FUNCTION_BLOCK Mc2AxisPTP_HMI EXTENDS HmiFunction
VAR
	Axis : I_Mc2Axis_PTP;
	{ attribute 'TcHmiSymbol.AddSymbol' }
	{ attribute 'TcHmiSymbol.AddSymbol.UserGroups' := '__SystemAdministrators,Admin' }
	AxisPTP_HMI : ST_AxisPTP_HMI;
END_VAR

PROPERTY ControlObject : I_Base
SET
__QueryInterface(ControlObject,Axis);
END_SET
END_PROPERTY

METHOD CyclicLogic
VAR_INST
	EnableRT	   : R_TRIG;
	DisableRT	   : R_TRIG;
	StopRT		   : R_TRIG;
	HomeRT		   : R_TRIG;
	ResetRT		   : R_TRIG;
	MoveAbsoluteRT : R_TRIG;
	MoveModuloRT   : R_TRIG;
	MoveRelativeRT : R_TRIG;
	MoveVelocityRT : R_TRIG;
END_VAR
IF Axis = 0 THEN
	RETURN;
END_IF

AxisPTP_HMI.HmiEnabled				  := Enabled;
AxisPTP_HMI.ActualAcceleration		  := Axis.ActualAcceleration;
AxisPTP_HMI.ActualPosition			  := Axis.ActualPosition;
AxisPTP_HMI.ActualPositionModulo	  := Axis.ActualPositionModulo;
AxisPTP_HMI.ActualTorque			  := Axis.ActualTorque;
AxisPTP_HMI.ActualVelocity			  := Axis.ActualVelocity;
AxisPTP_HMI.Busy					  := Axis.Busy;
AxisPTP_HMI.Error					  := Axis.Error;
AxisPTP_HMI.ErrorId					  := Axis.ErrorId;
AxisPTP_HMI.Name					  := Axis.Name;
AxisPTP_HMI.Status.Coupled			  := Axis.Axis.Status.Coupled;
AxisPTP_HMI.Status.Disabled			  := Axis.Axis.Status.Disabled;
AxisPTP_HMI.Status.SynchronizedMotion := Axis.Axis.Status.SynchronizedMotion;

// HMI Commands
StopRT(CLK := AxisPTP_HMI.Stop.Active);
IF StopRT.Q THEN
	IF AxisPTP_HMI.Stop.Permissive.OK THEN
		Axis.Stop();
	END_IF
END_IF

ResetRT(CLK := AxisPTP_HMI.Reset.Active);
IF ResetRT.Q THEN
	IF AxisPTP_HMI.Reset.Permissive.OK THEN
		Axis.Reset();
	END_IF
END_IF

IF Enabled THEN
	EnableRT(CLK := AxisPTP_HMI.Enable.Active);
	IF EnableRT.Q THEN
		IF AxisPTP_HMI.Enable.Permissive.OK THEN
			Axis.Enable();
		END_IF
	END_IF

	DisableRT(CLK := AxisPTP_HMI.Disable.Active);
	IF DisableRT.Q THEN
		IF AxisPTP_HMI.Disable.Permissive.OK THEN
			Axis.Disable();
		END_IF
	END_IF

	IF AxisPTP_HMI.JogBackwardSlow.Active THEN
		IF AxisPTP_HMI.JogBackwardSlow.Permissive.OK THEN
			Axis.JogMode := E_JogMode.MC_JOGMODE_STANDARD_SLOW;
			Axis.Jog(JogForward := FALSE, JogBackwards := TRUE);
		END_IF
	ELSIF AxisPTP_HMI.JogForwardSlow.Active THEN
		Axis.JogMode := E_JogMode.MC_JOGMODE_STANDARD_SLOW;
		Axis.Jog(JogForward := TRUE, JogBackwards := FALSE);
	ELSIF AxisPTP_HMI.JogBackwardFast.Active THEN
		Axis.JogMode := E_JogMode.MC_JOGMODE_STANDARD_FAST;
		Axis.Jog(JogForward := FALSE, JogBackwards := TRUE);
	ELSIF AxisPTP_HMI.JogForwardFast.Active THEN
		Axis.JogMode := E_JogMode.MC_JOGMODE_STANDARD_FAST;
		Axis.Jog(JogForward := TRUE, JogBackwards := FALSE);
	ELSE
		Axis.JogMode := E_JogMode.MC_JOGMODE_STANDARD_SLOW;
		Axis.Jog(JogForward := FALSE, JogBackwards := FALSE);
	END_IF

	HomeRT(CLK := AxisPTP_HMI.Home.Active);
	IF HomeRT.Q THEN
		IF AxisPTP_HMI.Home.Permissive.OK THEN
			Axis.Home();
		END_IF
	END_IF

	MoveAbsoluteRT(CLK := AxisPTP_HMI.MoveAbsolute.Active);
	IF MoveAbsoluteRT.Q THEN
		IF AxisPTP_HMI.MoveAbsolute.Permissive.OK THEN
			Axis.MoveAbsolute(AxisPTP_HMI.TargetPosition);
		END_IF
	END_IF

	MoveModuloRT(CLK := AxisPTP_HMI.MoveModulo.Active);
	IF MoveModuloRT.Q THEN
		IF AxisPTP_HMI.MoveModulo.Permissive.OK THEN
			Axis.MoveModulo(AxisPTP_HMI.TargetPosition);
		END_IF
	END_IF

	MoveRelativeRT(CLK := AxisPTP_HMI.MoveRelative.Active);
	IF MoveRelativeRT.Q THEN
		IF AxisPTP_HMI.MoveRelative.Permissive.OK THEN
			Axis.MoveRelative(AxisPTP_HMI.TargetDistance);
		END_IF
	END_IF

	MoveVelocityRT(CLK := AxisPTP_HMI.MoveVelocity.Active);
	IF MoveVelocityRT.Q THEN
		IF AxisPTP_HMI.MoveVelocity.Permissive.OK THEN
			Axis.MoveVelocity(AxisPTP_HMI.TargetVelocity);
		END_IF
	END_IF
END_IF
END_METHOD

PROPERTY DisablePermissive : I_Permissive
GET
DisablePermissive := AxisPTP_HMI.Disable.Permissive;
END_GET
END_PROPERTY

PROPERTY EnablePermissive : I_Permissive
GET
EnablePermissive := AxisPTP_HMI.Enable.Permissive;
END_GET
END_PROPERTY

(*FB_Init is always available implicitly and it is used primarily for initialization.
The return value is not evaluated. For a specific influence, you can also declare the
methods explicitly and provide additional code there with the standard initialization
code. You can evaluate the return value.*)
METHOD FB_Init : BOOL
VAR_INPUT
	(* TRUE: the retain variables are initialized (reset warm / reset cold)*)
	bInitRetains : BOOL;

	(* TRUE: the instance will be copied to the copy code afterward (online change)   *)
	bInCopyCode : BOOL;
	Name		: T_MaxString;
	Axis		: I_Mc2Axis_PTP;
	Unit		: STRING;
END_VAR
THIS^.Axis		 := Axis;
ControlType		 := 'AxisPTP';
LinkObject		 := 'AxisPTP_HMI';
AxisPTP_HMI.Unit := Unit;
END_METHOD

PROPERTY HomePermissive : I_Permissive
GET
HomePermissive := AxisPTP_HMI.Home.Permissive;
END_GET
END_PROPERTY

PROPERTY JogBackwardFastPermissive : I_Permissive
GET
JogBackwardFastPermissive := AxisPTP_HMI.JogBackwardFast.Permissive;
END_GET
END_PROPERTY

PROPERTY JogBackwardSlowPermissive : I_Permissive
GET
JogBackwardSlowPermissive := AxisPTP_HMI.JogBackwardSlow.Permissive;
END_GET
END_PROPERTY

PROPERTY JogForwardFastPermissive : I_Permissive
GET
JogForwardFastPermissive := AxisPTP_HMI.JogForwardFast.Permissive;
END_GET
END_PROPERTY

PROPERTY JogForwardSlowPermissive : I_Permissive
GET
JogForwardSlowPermissive := AxisPTP_HMI.JogForwardSlow.Permissive;
END_GET
END_PROPERTY

PROPERTY MoveAbsolutePermissive : I_Permissive
GET
MoveAbsolutePermissive := AxisPTP_HMI.MoveAbsolute.Permissive;
END_GET
END_PROPERTY

PROPERTY MoveModuloPermissive : I_Permissive
GET
MoveModuloPermissive := AxisPTP_HMI.MoveModulo.Permissive;
END_GET
END_PROPERTY

PROPERTY MoveRelativePermissive : I_Permissive
GET
MoveRelativePermissive := AxisPTP_HMI.MoveRelative.Permissive;
END_GET
END_PROPERTY

PROPERTY MoveVelocityPermissive : I_Permissive
GET
MoveVelocityPermissive := AxisPTP_HMI.MoveVelocity.Permissive;
END_GET
END_PROPERTY

PROPERTY ResetPermissive : I_Permissive
GET
ResetPermissive := AxisPTP_HMI.Reset.Permissive;
END_GET
END_PROPERTY

PROPERTY StopPermissive : I_Permissive
GET
StopPermissive := AxisPTP_HMI.Stop.Permissive;
END_GET
END_PROPERTY

END_FUNCTION_BLOCK

(* stored: Version 1.1.0.1, ProductVersion 3.1.4026.20
   POU Mc2AxisPTP_HMI: Id {e48832af-14b2-499a-a3f7-17b5e3c2c043}, SpecialFunc None
   Folder Button Permissives: Id {ec4ff6f5-3915-469b-989a-722f4eeac77c}
   Property ControlObject: Id {6f5fdd79-a376-4b59-a654-75185406e984}
   Set Set: Id {87e8668b-dfba-4f7d-a8bd-473573b71a68}
   Method CyclicLogic: Id {9e4a2d0b-42d1-4a3f-bfe7-bcbc4b120734}
   Property DisablePermissive: Id {b2e57bab-a249-4965-81c9-49b9ce365ac1}
   Get Get: Id {1ffe4964-8e18-45db-ae65-a9a5c34fe5a4}
   Property EnablePermissive: Id {a5d9222e-c7da-482c-937e-cf94323f91c7}
   Get Get: Id {c9889fb7-d31f-48d8-8ecb-44f007914b8c}
   Method FB_Init: Id {6a5bd057-7513-4b13-9e46-c42c8fb6c16e}
   Property HomePermissive: Id {2d45b464-ae39-4613-ab1d-8e8438be2ac3}
   Get Get: Id {d7f24ff6-8858-4a39-84ec-06d9af61ac59}
   Property JogBackwardFastPermissive: Id {fa6f30d9-7408-4c95-822a-38bf91c7c423}
   Get Get: Id {cd04e466-bbc7-4567-af4c-9f7ab559d108}
   Property JogBackwardSlowPermissive: Id {b5f10fff-0dfe-4027-8428-697e8c5a567c}
   Get Get: Id {7f0e3e50-31d4-49c0-98a5-7c49a1db17bd}
   Property JogForwardFastPermissive: Id {88deac7e-b512-477c-82a8-dc8aa300f612}
   Get Get: Id {dafff7d6-8ff0-495d-bc79-b2a24d3666c5}
   Property JogForwardSlowPermissive: Id {ecc504b2-e3af-4830-bac5-afe34b2f6bc3}
   Get Get: Id {0a184746-52f3-442d-ae5a-7963f9f5f2e7}
   Property MoveAbsolutePermissive: Id {797188eb-4d0d-4eba-8c92-f2c7c93698ef}
   Get Get: Id {7bd98e37-1a94-4b7b-ad05-ba6a9f438fb9}
   Property MoveModuloPermissive: Id {fb927034-2c38-442d-990c-f0df03dd223e}
   Get Get: Id {d9ecdbbc-505c-4b15-9867-4da6624b67f9}
   Property MoveRelativePermissive: Id {743468ad-f4ce-4f61-bae9-0c0d01ee8683}
   Get Get: Id {11f4fb1b-9bc7-4f41-b111-54d07cf01618}
   Property MoveVelocityPermissive: Id {10cb4381-af8c-401f-9663-a950fcab4579}
   Get Get: Id {278dfc60-857f-4a95-9a0b-db3e3b5791d6}
   Property ResetPermissive: Id {d09bb902-1471-4a4d-91ca-9d2851188990}
   Get Get: Id {d6d63940-2c34-4a78-832b-abf634cd9c76}
   Property StopPermissive: Id {0561ba9c-b6a4-408a-87bd-99373376dac9}
   Get Get: Id {89b12035-e84a-4acc-b61e-f5cb8be11b9e} *)
